(* CODESYS project Proje_2.project
   Title: Step
   Version: 0.0.0.0
   Author: MustafaZahid

Project tree, tasks and I/O mapping:
  MyController : TM241C24T/U, Schneider Electric, order no. TM241C24T/U, version 4.0.6.18
    application Application
      task MAST (cyclic, interval 20 ms, priority 15, watchdog 100 ms x 1) calls POU
      global variables GVL
      program POU [LD]
      FunctionBlocks/
        function block Motor_Administration [LD]
        function block Axis_Configuration [LD]
        function block Set_To_Reset [LD]
    DI : Digital Inputs, Schneider Electric, version 4.0.6.18
        input  iwDI_IW0 : WORD  // IW0
        input  ibDI_IB1 : BYTE  // IB1
    DQ : Digital Outputs, Schneider Electric, version 4.0.6.18
        settings: Outputs Usage = 3
        output qwDQ_QW0 : WORD  // QW0
        output qbDQ_QB1 : BYTE  // QB1
    Counters : Counters, Schneider Electric, version 4.0.6.18
    Pulse_Generators : Pulse Generators, Schneider Electric, version 4.0.6.18
        settings: Instance name = 'Axis_1'; PROBE input History = 'old=0 new=-1'; REF input History = 'old=0 new=-1'; B output History = 'old=-1 new=1'; A output History = 'old=-1 new=0'; Temporary Instance name = 'Axis_1'
    Cartridge_1 : Cartridge, Schneider Electric, version 4.0.6.18
    IO_Bus : IO bus - TM3, Schneider Electric, version 4.0.6.18
    COM_Bus : COM bus, Schneider Electric, version 4.0.6.18
    Serial_Line_1 : Serial line, Schneider Electric, version 4.0.6.18
      SoMachine_Network_Manager : SoMachine-Network Manager, Schneider Electric, version 4.0.0.2
    Serial_Line_2 : Serial line, Schneider Electric, version 4.0.6.18
      Modbus_Manager : Modbus Manager, Schneider Electric, version 4.0.0.2
  text list GlobalTextList
*)

// MyController/Application/GVL
VAR_GLOBAL
	Power_En: BOOL;
	Homing_En: BOOL;
	Reset_En: BOOL;
	Stop_En: BOOL;
	MoveToBending_En: BOOL;
	MoveToHome_En: BOOL;
	Sensor_Detected: BOOL;
	ActualPosition: DINT;
	HomingDone: BOOL;
	ResetDone: BOOL;
END_VAR

// MyController/Application/POU
PROGRAM POU
VAR
	Motor_Administration_0: Motor_Administration;
	Axis_Config: Axis_Configuration;
	Timer_1: TON;
	Timer_2: TON;
	BendingMachine: BOOL;
	CTU_0: CTU;
END_VAR
VAR // added by the converter: edge detectors and wires of the graphical bodies
    _w1 : BOOL;
    _rt1 : R_TRIG;
END_VAR

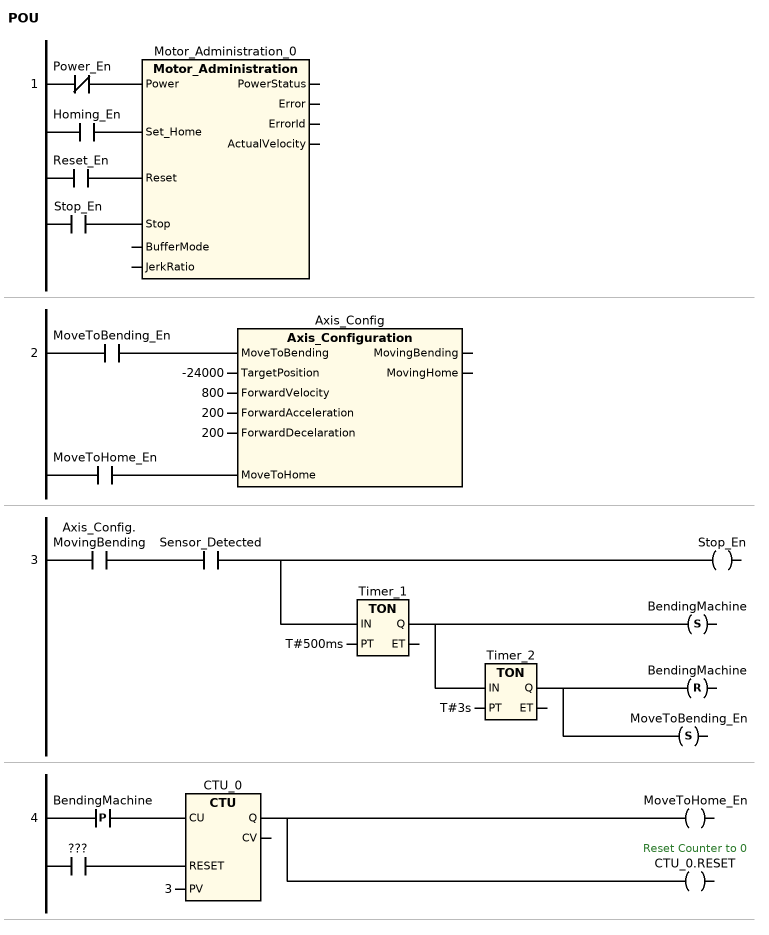
// NETWORK 1
Motor_Administration_0(Power := NOT Power_En, Set_Home := Homing_En, Reset := Reset_En, Stop := Stop_En); // Motor_Administration

// NETWORK 2
Axis_Config(
    MoveToBending := MoveToBending_En,
    TargetPosition := -24000,
    ForwardVelocity := 800,
    ForwardAcceleration := 200,
    ForwardDecelaration := 200,
    MoveToHome := MoveToHome_En); // Axis_Configuration

// NETWORK 3
_w1 := Axis_Config.MovingBending AND Sensor_Detected;
Stop_En := _w1;
Timer_1(IN := _w1, PT := T#500ms); // TON
BendingMachine S= Timer_1.Q;
Timer_2(IN := Timer_1.Q, PT := T#3s); // TON
BendingMachine R= Timer_2.Q;
MoveToBending_En S= Timer_2.Q;

// NETWORK 4
//   CTU_0.RESET: Reset Counter to 0
_rt1(CLK := BendingMachine);
CTU_0(CU := _rt1.Q, PV := 3); // CTU
MoveToHome_En := CTU_0.Q;
CTU_0.RESET := CTU_0.Q;

END_PROGRAM

// MyController/Application/FunctionBlocks/Motor_Administration
FUNCTION_BLOCK Motor_Administration
VAR_INPUT
	Power: BOOL;
	Set_Home: BOOL;
	Reset: BOOL;
	Stop: BOOL;
	BufferMode: MC_BUFFER_MODE;
	JerkRatio: INT;
END_VAR
VAR_OUTPUT
	PowerStatus: BOOL;
	Error: BOOL;
	ErrorId: PTO_ERROR;
	ActualVelocity: DINT;
END_VAR
VAR
	MC_Power: MC_Power_PTO;
	MC_Home: MC_Home_PTO;
	MC_Reset: MC_Reset_PTO;
	MC_Stop: MC_Stop_PTO;
	MC_SetPosition: MC_SetPosition_PTO;
	MC_ReadActualPosition: MC_ReadActualPosition_PTO;
	MC_MoveAbsolute: MC_MoveAbsolute_PTO;
	MC_ReadActualVelocity: MC_ReadActualVelocity_PTO;
END_VAR

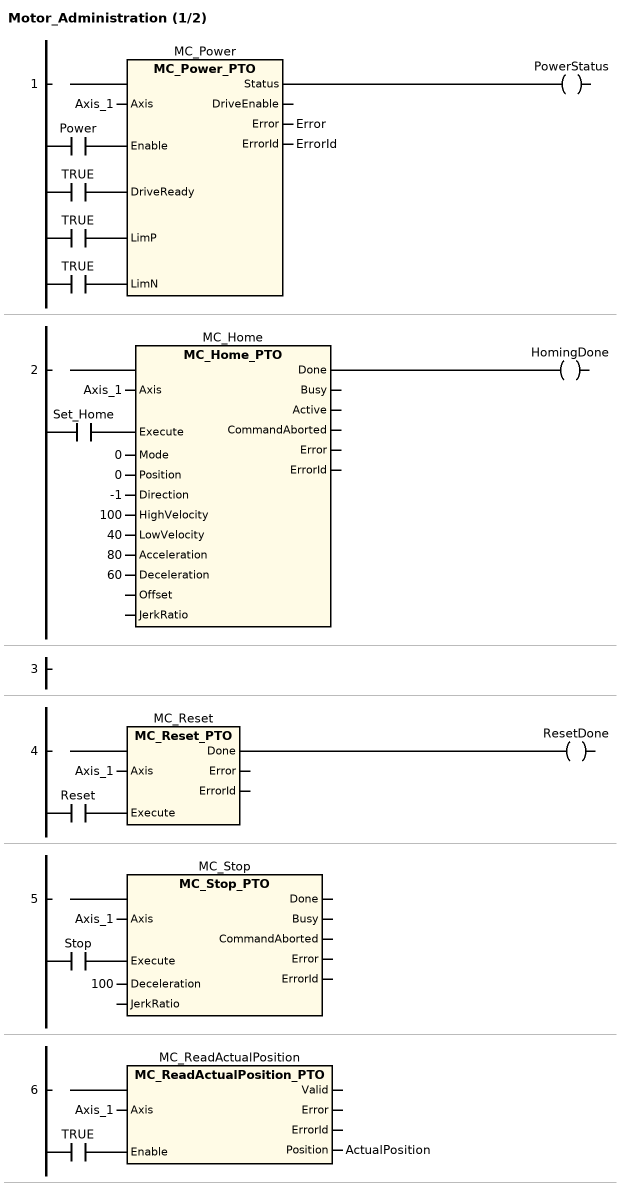
// NETWORK 1
MC_Power(
    Axis := Axis_1,
    Enable := Power,
    DriveReady := TRUE,
    LimP := TRUE,
    LimN := TRUE,
    Error => Error,
    ErrorId => ErrorId); // MC_Power_PTO
PowerStatus := MC_Power.Status;

// NETWORK 2
MC_Home(
    Axis := Axis_1,
    Execute := Set_Home,
    Mode := 0,
    Position := 0,
    Direction := -1,
    HighVelocity := 100,
    LowVelocity := 40,
    Acceleration := 80,
    Deceleration := 60); // MC_Home_PTO
HomingDone := MC_Home.Done;

// NETWORK 3

// NETWORK 4
MC_Reset(Axis := Axis_1, Execute := Reset); // MC_Reset_PTO
ResetDone := MC_Reset.Done;

// NETWORK 5
MC_Stop(Axis := Axis_1, Execute := Stop, Deceleration := 100); // MC_Stop_PTO

// NETWORK 6
MC_ReadActualPosition(Axis := Axis_1, Enable := TRUE, Position => ActualPosition); // MC_ReadActualPosition_PTO

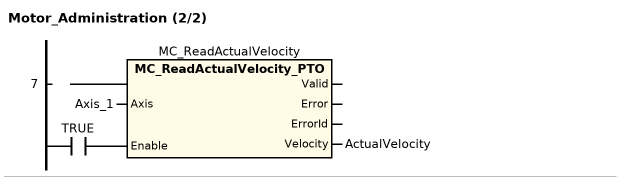
// NETWORK 7
MC_ReadActualVelocity(Axis := Axis_1, Enable := TRUE, Velocity => ActualVelocity); // MC_ReadActualVelocity_PTO

END_FUNCTION_BLOCK

// MyController/Application/FunctionBlocks/Axis_Configuration
FUNCTION_BLOCK Axis_Configuration
VAR_INPUT
	MoveToBending: BOOL;
	TargetPosition: DINT;
	ForwardVelocity: DINT;
	ForwardAcceleration: DINT;
	ForwardDecelaration: DINT;
	MoveToHome: BOOL;
END_VAR
VAR_OUTPUT
	MovingBending: BOOL;
	MovingHome: BOOL;
END_VAR
VAR
	MC_Absolute_Positive: MC_MoveAbsolute_PTO;
	MC_Absolute_Negative: MC_MoveAbsolute_PTO;
	Positive: BOOL;
	Negative: BOOL;
END_VAR
VAR // added by the converter: edge detectors and wires of the graphical bodies
    _rt1, _rt2 : R_TRIG;
END_VAR

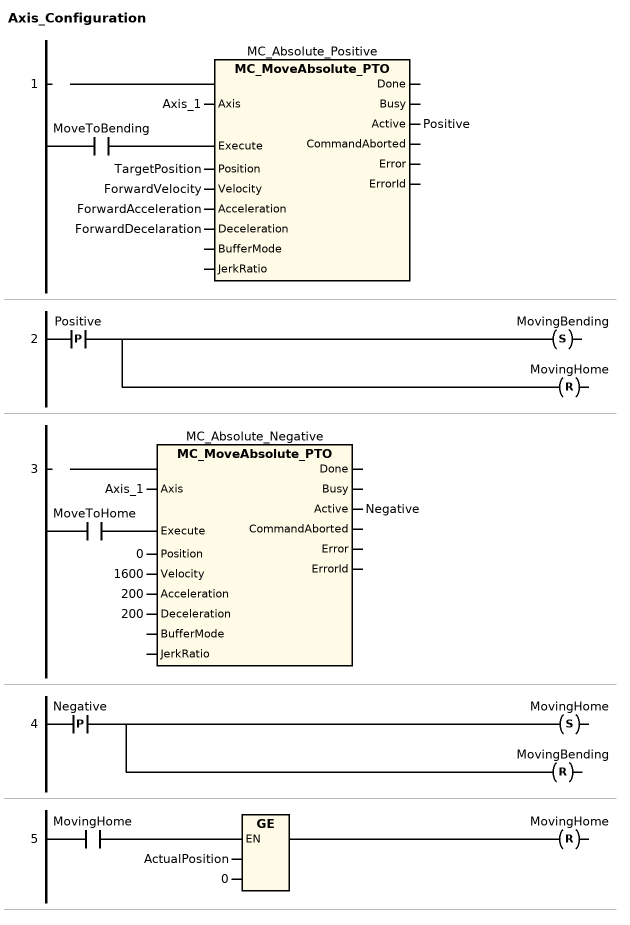
// NETWORK 1
MC_Absolute_Positive(
    Axis := Axis_1,
    Execute := MoveToBending,
    Position := TargetPosition,
    Velocity := ForwardVelocity,
    Acceleration := ForwardAcceleration,
    Deceleration := ForwardDecelaration,
    Active => Positive); // MC_MoveAbsolute_PTO

// NETWORK 2
_rt1(CLK := Positive);
MovingBending S= _rt1.Q;
MovingHome R= _rt1.Q;

// NETWORK 3
MC_Absolute_Negative(
    Axis := Axis_1,
    Execute := MoveToHome,
    Position := 0,
    Velocity := 1600,
    Acceleration := 200,
    Deceleration := 200,
    Active => Negative); // MC_MoveAbsolute_PTO

// NETWORK 4
_rt2(CLK := Negative);
MovingHome S= _rt2.Q;
MovingBending R= _rt2.Q;

// NETWORK 5
MovingHome R= MovingHome AND ActualPosition >= 0;

END_FUNCTION_BLOCK

// MyController/Application/FunctionBlocks/Set_To_Reset
FUNCTION_BLOCK Set_To_Reset
VAR_INPUT
END_VAR
VAR_OUTPUT
END_VAR
VAR
	Timer: TON;
END_VAR

VAR_IN_OUT
	Input: BOOL;
END_VAR

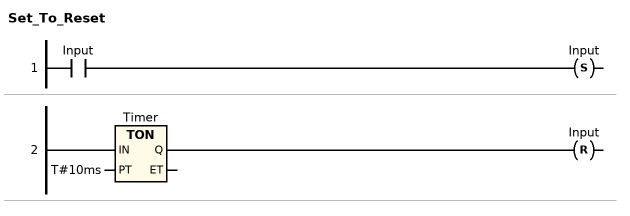
// NETWORK 1
Input S= Input;

// NETWORK 2
Timer(IN := TRUE, PT := T#10ms); // TON
Input R= Timer.Q;

END_FUNCTION_BLOCK
